// TwinCAT 3 PLC project PRG_Test_MachineControl
// ProgramVersion: 3.1.4024.0
// libraries:
//   B_Base, * (RafalOS)
//   B_IO, * (RafalOS)
//   B_MachineControl, * (RafalOS)
//   B_StatesAndModes, * (RafalOS)
//   Tc2_Standard, * (Beckhoff Automation GmbH)
//   Tc2_System, * (Beckhoff Automation GmbH)
//   Tc3_Module, * (Beckhoff Automation GmbH)
//   TcUnit, * (www.tcunit.org)
// project tree:
//   GVLs/ GVL_TopElement1.TcGVL (not stored), GVL_TopElement2.TcGVL (not stored), GVL_Variable.TcGVL
//   / PlcTask.TcTTO
//   POUs/ FB_MachineControlTest.TcPOU, FB_MyNewConfiguration.TcPOU
//   POUs/POUs TopElement1/ FB_ControlElement1.TcPOU, FB_ControlElement2.TcPOU, FB_TopElement1.TcPOU, ITF_ControlElement1.TcIO, ITF_ControlElement2.TcIO, ITF_TopElement1.TcIO
//   POUs/POUs TopElement2/ FB_ControlElement3.TcPOU, FB_ControlElement5.TcPOU (not stored), FB_ControlElement4.TcPOU, FB_ControlElement6.TcPOU (not stored), FB_GroupElement1.TcPOU (not stored), FB_TopElement2.TcPOU, ITF_ControlElement3.TcIO, ITF_ControlElement5.TcIO, ITF_ControlElement4.TcIO (not stored), ITF_ControlElement6.TcIO (not stored), ITF_GroupElement1.TcIO, ITF_TopElement2.TcIO
//   TESTs/ PRG_Test.TcPOU
// real-time tasks:
//   TASK PlcTask: cycle T#10ms, priority 20, ADS port 350

CONFIGURATION PRG_Test_MachineControl
    RESOURCE PLC ON TwinCAT3
        TASK PlcTask(INTERVAL := T#10ms, PRIORITY := 20);
        PROGRAM PRG_Test WITH PlcTask : PRG_Test;
    END_RESOURCE
END_CONFIGURATION

// ---- GVLs/GVL_Variable.TcGVL
{attribute 'qualified_only'}
VAR_GLOBAL
	fbMyNewConfiguration		: FB_MyNewConfiguration;
	
(* zmienne potrzebne do przetestowania samego SaMController	*)
	fbTime						: FB_BaseTime;
	fbLocation					: FB_BaseLocation;
	fbLogger					: FB_BaseLogger;
	stCommonData				: ST_BaseCommonData;
	flSS1						: FB_BaseFlag;
	flSTO						: FB_BaseFlag;
	fbMySaMController			: FB_SaMController;
END_VAR

// ---- POUs/POUs TopElement1/ITF_ControlElement1.TcIO
INTERFACE ITF_ControlElement1 EXTENDS ITF_BaseControlElement

END_INTERFACE

// ---- POUs/POUs TopElement1/ITF_ControlElement2.TcIO
INTERFACE ITF_ControlElement2 EXTENDS ITF_BaseControlElement

END_INTERFACE

// ---- POUs/POUs TopElement1/ITF_TopElement1.TcIO
INTERFACE ITF_TopElement1 EXTENDS ITF_BaseTopElement

END_INTERFACE

// ---- POUs/POUs TopElement2/ITF_ControlElement3.TcIO
INTERFACE ITF_ControlElement3 EXTENDS ITF_BaseControlElement

END_INTERFACE

// ---- POUs/POUs TopElement2/ITF_ControlElement5.TcIO
INTERFACE ITF_ControlElement5 EXTENDS ITF_BaseControlElement

END_INTERFACE

// ---- POUs/POUs TopElement2/ITF_GroupElement1.TcIO
INTERFACE ITF_GroupElement1 EXTENDS ITF_BaseGroupElement

END_INTERFACE

// ---- POUs/POUs TopElement2/ITF_TopElement2.TcIO
INTERFACE ITF_TopElement2 EXTENDS ITF_BaseTopElement

END_INTERFACE

// ---- TESTs/PRG_Test.TcPOU
PROGRAM PRG_Test
VAR
	fbSaMControllerTest				: FB_SaMControllerTest;
	fbMachineControlTest			: FB_MachineControl_NoneTE_Test;
	
END_VAR


	TcUnit.RUN_IN_SEQUENCE ();

END_PROGRAM

// ---- POUs/FB_MyNewConfiguration.TcPOU
FUNCTION_BLOCK FB_MyNewConfiguration EXTENDS FB_Base IMPLEMENTS ITF_Configuration
VAR

END_VAR

METHOD AddTopElementToLogger : BOOL
GVL_TopElement1.fbTopElement1.JoinTheLogger ();
GVL_TopElement2.fbTopElement2.JoinTheLogger ();
END_METHOD

(*			
	EVERDE sp. z o.o.
	Rafał Osajda		29.10.2025		TC 4024.66
	Dodawanie TopElementu do systemu
*)
METHOD AddTopElementToMachineControl : BOOL
VAR_INPUT
	itfMachineControl	: B_MachineControl.ITF_MachineControlConfigure;
END_VAR
THIS^.SetText (eLocation := E_BaseLocation.pl, wsDescription := "TopElement 1 pl");
THIS^.SetText (eLocation := E_BaseLocation.en, wsDescription := "TopElement 1 en");
THIS^.SetText (eLocation := E_BaseLocation.de, wsDescription := "TopElement 1 de");
GVL_TopElement1.fbTopElement1.SetName (stName := THIS^.GetTexts ());
itfMachineControl.AddTopElementFromConfiguration (fbTopElement	:= GVL_TopElement1.fbTopElement1);

THIS^.SetText (eLocation := E_BaseLocation.pl, wsDescription := "TopElement 2 pl");
THIS^.SetText (eLocation := E_BaseLocation.en, wsDescription := "TopElement 2 en");
THIS^.SetText (eLocation := E_BaseLocation.de, wsDescription := "TopElement 2 de");
GVL_TopElement1.fbTopElement1.SetName (stName := THIS^.GetTexts ());
itfMachineControl.AddTopElementFromConfiguration (fbTopElement	:= GVL_TopElement2.fbTopElement2);
END_METHOD

{warning 'add method implementation '}
METHOD SetStartMode : BOOL
VAR_INPUT
	itfMachineControl	: B_MachineControl.ITF_MachineControlConfigure;
END_VAR
END_METHOD

METHOD StateAndModes : BOOL
VAR_INPUT
	itfMachineControl	: B_MachineControl.ITF_MachineControlConfigure;
END_VAR
END_METHOD

END_FUNCTION_BLOCK

// ---- POUs/FB_MachineControlTest.TcPOU
FUNCTION_BLOCK FB_MachineControlTest EXTENDS TcUnit.FB_TestSuite
VAR

END_VAR


T01_TestPierwszegoPrzejscia ();
T02_TestInicjalizacjiSaM ();

METHOD PROTECTED T01_TestPierwszegoPrzejscia
VAR_INPUT
END_VAR
IF (TcUnit.TEST_ORDERED ('T01_TestPierwszegoPrzejscia')) THEN
	PRG_SystemControlMachineInit ();	//<- do prawdziwego programu
	AssertEquals_INT (Expected := 0, Actual := GVL_SystemVariable.fbMachineConfigure.iNubmerOfAddedConfigure, Message := 'T01_01 - blad ilosci konfiguracji');

	GVL_SystemVariable.fbMachineConfigure.AddConfiguration (fbConfigure := GVL_Variable.fbMyNewConfiguration); 		//<- do prawdziwego programu
	AssertEquals_INT (Expected := 1, Actual := GVL_SystemVariable.fbMachineConfigure.iNubmerOfAddedConfigure, Message := 'T01_02 - blad ilosci konfiguracji');

	PRG_SystemControlMachineWork ();		//<- do prawdziwego programu
	AssertTrue (Condition := GVL_SystemVariable.fbMachineControl.bInitializeCycle, Message := 'T02_01 - blad pierwszego przejscia');
	AssertTrue (Condition := GVL_SystemVariable.fbMachineControl.bInitDone, Message := 'T02_02 - blad inicjalizacji');
	AssertEquals_UINT (Expected := 20, Actual := GVL_SystemVariable.fbLogger.uiNumerOfReportsIntheSystem, Message := 'T02_03 - Bledna ilosc zgloszen');
	AssertEquals_UINT (Expected := 34, Actual := GVL_SystemVariable.fbMachineControl.uiNumberOfAllAddedElements, Message := 'T02_04 - bledna ilosc elementow');
	
	
	
	TcUnit.TEST_FINISHED ();
END_IF
END_METHOD

METHOD PROTECTED T02_TestInicjalizacjiSaM
VAR
	
END_VAR
IF (TcUnit.TEST_ORDERED ('T02_TestInicjalizacjiSaM')) THEN
	GVL_Variable.stCommonData.itfTime			:= GVL_Variable.fbTime;
	GVL_Variable.stCommonData.itfLocaciotn		:= GVL_Variable.fbLocation;
	GVL_Variable.stCommonData.itfLogger			:= GVL_Variable.fbLogger;
	GVL_Variable.fbMySaMController.LinkCommonData (stCommonData := GVL_Variable.stCommonData);
	GVL_Variable.fbMySaMController.LinkSS1 (fbSS1	:= GVL_Variable.flSS1);
	GVL_Variable.fbMySaMController.LinkSTO (fbSTO	:= GVL_Variable.flSTO);
	
	TcUnit.TEST_FINISHED ();
END_IF
END_METHOD

END_FUNCTION_BLOCK

// ---- POUs/POUs TopElement1/FB_ControlElement1.TcPOU
FUNCTION_BLOCK FB_ControlElement1 EXTENDS FB_BaseControlElement IMPLEMENTS ITF_ControlElement1
VAR
	
	itfsenStart			: ITF_IOSensor;
	itfsenEnd			: ITF_IOSensor;	
END_VAR

METHOD FB_init : BOOL
VAR_INPUT
	bInitRetains : BOOL; // if TRUE, the retain variables are initialized (warm start / cold start)
	bInCopyCode : BOOL;  // if TRUE, the instance afterwards gets moved into the copy code (online change)
	itfsenStart			: ITF_IOSensor;
	itfsenEnd			: ITF_IOSensor;	
	
END_VAR
THIS^.itfsenStart					:= itfsenStart;
THIS^.AddComponent (itfComponent	:= itfsenStart);
THIS^.SetText (eLocation 			:= E_BaseLocation.pl, wsDescription := "Nazwa komponentu 1 pl");
THIS^.SetText (eLocation 			:= E_BaseLocation.en, wsDescription := "Nazwa komponentu 1 en");
THIS^.SetText (eLocation 			:= E_BaseLocation.de, wsDescription := "Nazwa komponentu 1 de");
THIS^.itfsenStart.SetName (stName	:= THIS^.GetTexts ());

THIS^.itfsenEnd						:= itfsenEnd;
THIS^.AddComponent (itfComponent	:= itfsenEnd);
THIS^.SetText (eLocation 			:= E_BaseLocation.pl, wsDescription := "Nazwa komponentu 2 pl");
THIS^.SetText (eLocation 			:= E_BaseLocation.en, wsDescription := "Nazwa komponentu 2 en");
THIS^.SetText (eLocation 			:= E_BaseLocation.de, wsDescription := "Nazwa komponentu 2 de");
THIS^.itfsenEnd.SetName (stName	:= THIS^.GetTexts ());
END_METHOD

END_FUNCTION_BLOCK

// ---- POUs/POUs TopElement1/FB_ControlElement2.TcPOU
FUNCTION_BLOCK FB_ControlElement2 EXTENDS FB_BaseControlElement IMPLEMENTS ITF_ControlElement2
VAR
	
	itfsenStart			: ITF_IOSensor;
	itfsenEnd			: ITF_IOSensor;	
	itfsenPosition1		: ITF_IOSensor;	
	itfsenPosition2		: ITF_IOSensor;	
END_VAR

METHOD FB_init : BOOL
VAR_INPUT
	bInitRetains : BOOL; // if TRUE, the retain variables are initialized (warm start / cold start)
	bInCopyCode : BOOL;  // if TRUE, the instance afterwards gets moved into the copy code (online change)
	itfsenStart			: ITF_IOSensor;
	itfsenEnd			: ITF_IOSensor;	
	itfsenPosition1		: ITF_IOSensor;	
	itfsenPosition2		: ITF_IOSensor;	
END_VAR
THIS^.itfsenStart					:= itfsenStart;
THIS^.AddComponent (itfComponent	:= itfsenStart);
THIS^.SetText (eLocation 			:= E_BaseLocation.pl, wsDescription := "Nazwa komponentu 1 pl");
THIS^.SetText (eLocation 			:= E_BaseLocation.en, wsDescription := "Nazwa komponentu 1 en");
THIS^.SetText (eLocation 			:= E_BaseLocation.de, wsDescription := "Nazwa komponentu 1 de");
THIS^.itfsenStart.SetName (stName	:= THIS^.GetTexts ());

THIS^.itfsenEnd						:= itfsenEnd;
THIS^.AddComponent (itfComponent	:= itfsenEnd);
THIS^.SetText (eLocation 			:= E_BaseLocation.pl, wsDescription := "Nazwa komponentu 2 pl");
THIS^.SetText (eLocation 			:= E_BaseLocation.en, wsDescription := "Nazwa komponentu 2 en");
THIS^.SetText (eLocation 			:= E_BaseLocation.de, wsDescription := "Nazwa komponentu 2 de");
THIS^.itfsenEnd.SetName (stName	:= THIS^.GetTexts ());

THIS^.itfsenPosition1				:= itfsenPosition1;
THIS^.AddComponent (itfComponent	:= itfsenPosition1);
THIS^.SetText (eLocation 			:= E_BaseLocation.pl, wsDescription := "Nazwa komponentu 3 pl");
THIS^.SetText (eLocation 			:= E_BaseLocation.en, wsDescription := "Nazwa komponentu 3 en");
THIS^.SetText (eLocation 			:= E_BaseLocation.de, wsDescription := "Nazwa komponentu 3 de");
THIS^.itfsenPosition1.SetName (stName	:= THIS^.GetTexts ());

THIS^.itfsenPosition2				:= itfsenPosition2;
THIS^.AddComponent (itfComponent	:= itfsenPosition2);
THIS^.SetText (eLocation 			:= E_BaseLocation.pl, wsDescription := "Nazwa komponentu 4 pl");
THIS^.SetText (eLocation 			:= E_BaseLocation.en, wsDescription := "Nazwa komponentu 4 en");
THIS^.SetText (eLocation 			:= E_BaseLocation.de, wsDescription := "Nazwa komponentu 4 de");
THIS^.itfsenPosition2.SetName (stName	:= THIS^.GetTexts ());
END_METHOD

END_FUNCTION_BLOCK

// ---- POUs/POUs TopElement1/FB_TopElement1.TcPOU
FUNCTION_BLOCK FB_TopElement1 EXTENDS FB_BaseTopElement IMPLEMENTS ITF_TopElement1
VAR
	itfControlElement1		: ITF_ControlElement1;
	itfControlElement2		: ITF_ControlElement2;
	itfsenElementPosition1	: ITF_IOSensor;
	itfsenElementPosition2	: ITF_IOSensor;
END_VAR

METHOD FB_init : BOOL
VAR_INPUT
	bInitRetains : BOOL; // if TRUE, the retain variables are initialized (warm start / cold start)
	bInCopyCode : BOOL;  // if TRUE, the instance afterwards gets moved into the copy code (online change)
	itfControlElement1		: ITF_ControlElement1;
	itfControlElement2		: ITF_ControlElement2;
	itfsenElementPosition1	: ITF_IOSensor;
	itfsenElementPosition2	: ITF_IOSensor;
END_VAR
THIS^.itfControlElement1			:= itfControlElement1;
THIS^.AddComponent (itfComponent	:= itfControlElement1);
THIS^.SetText (eLocation 			:= E_BaseLocation.pl, wsDescription := "Nazwa controlelementu 1 pl");
THIS^.SetText (eLocation 			:= E_BaseLocation.en, wsDescription := "Nazwa controlelementu 1 en");
THIS^.SetText (eLocation 			:= E_BaseLocation.de, wsDescription := "Nazwa controlelementu 1 de");
THIS^.itfControlElement1.SetName (stName	:= THIS^.GetTexts ());

THIS^.itfControlElement2			:= itfControlElement2;
THIS^.AddComponent (itfComponent	:= itfControlElement2);
THIS^.SetText (eLocation 			:= E_BaseLocation.pl, wsDescription := "Nazwa controlelementu 2 pl");
THIS^.SetText (eLocation 			:= E_BaseLocation.en, wsDescription := "Nazwa controlelementu 2 en");
THIS^.SetText (eLocation 			:= E_BaseLocation.de, wsDescription := "Nazwa controlelementu 2 de");
THIS^.itfControlElement2.SetName (stName	:= THIS^.GetTexts ());

THIS^.itfsenElementPosition1		:= itfsenElementPosition1;
THIS^.AddComponent (itfComponent	:= itfsenElementPosition1);
THIS^.SetText (eLocation 			:= E_BaseLocation.pl, wsDescription := "Nazwa komponentu 1 pl");
THIS^.SetText (eLocation 			:= E_BaseLocation.en, wsDescription := "Nazwa komponentu 1 en");
THIS^.SetText (eLocation 			:= E_BaseLocation.de, wsDescription := "Nazwa komponentu 1 de");
THIS^.itfsenElementPosition1.SetName (stName	:= THIS^.GetTexts ());

THIS^.itfsenElementPosition2		:= itfsenElementPosition2;
THIS^.AddComponent (itfComponent	:= itfsenElementPosition2);
THIS^.SetText (eLocation 			:= E_BaseLocation.pl, wsDescription := "Nazwa komponentu 2 pl");
THIS^.SetText (eLocation 			:= E_BaseLocation.en, wsDescription := "Nazwa komponentu 2 en");
THIS^.SetText (eLocation 			:= E_BaseLocation.de, wsDescription := "Nazwa komponentu 2 de");
THIS^.itfsenElementPosition2.SetName (stName	:= THIS^.GetTexts ());
END_METHOD

END_FUNCTION_BLOCK

// ---- POUs/POUs TopElement2/FB_ControlElement3.TcPOU
FUNCTION_BLOCK FB_ControlElement3 EXTENDS FB_BaseControlElement IMPLEMENTS ITF_ControlElement3
VAR
	
	itfsenStart			: ITF_IOSensor;
	itfsenEnd			: ITF_IOSensor;	
END_VAR

METHOD FB_init : BOOL
VAR_INPUT
	bInitRetains : BOOL; // if TRUE, the retain variables are initialized (warm start / cold start)
	bInCopyCode : BOOL;  // if TRUE, the instance afterwards gets moved into the copy code (online change)
	itfsenStart			: ITF_IOSensor;
	itfsenEnd			: ITF_IOSensor;	
	
END_VAR
THIS^.itfsenStart					:= itfsenStart;
THIS^.AddComponent (itfComponent	:= itfsenStart);
THIS^.SetText (eLocation 			:= E_BaseLocation.pl, wsDescription := "Nazwa komponentu 1 pl");
THIS^.SetText (eLocation 			:= E_BaseLocation.en, wsDescription := "Nazwa komponentu 1 en");
THIS^.SetText (eLocation 			:= E_BaseLocation.de, wsDescription := "Nazwa komponentu 1 de");
THIS^.itfsenStart.SetName (stName	:= THIS^.GetTexts ());

THIS^.itfsenEnd						:= itfsenEnd;
THIS^.AddComponent (itfComponent	:= itfsenEnd);
THIS^.SetText (eLocation 			:= E_BaseLocation.pl, wsDescription := "Nazwa komponentu 2 pl");
THIS^.SetText (eLocation 			:= E_BaseLocation.en, wsDescription := "Nazwa komponentu 2 en");
THIS^.SetText (eLocation 			:= E_BaseLocation.de, wsDescription := "Nazwa komponentu 2 de");
THIS^.itfsenEnd.SetName (stName	:= THIS^.GetTexts ());
END_METHOD

END_FUNCTION_BLOCK

// ---- POUs/POUs TopElement2/FB_ControlElement4.TcPOU
FUNCTION_BLOCK FB_ControlElement4 EXTENDS FB_BaseControlElement IMPLEMENTS ITF_ControlElement4
VAR
	
	itfsenStart			: ITF_IOSensor;
	itfsenEnd			: ITF_IOSensor;	
	itfsenPosition1		: ITF_IOSensor;	
	itfsenPosition2		: ITF_IOSensor;	
END_VAR

METHOD FB_init : BOOL
VAR_INPUT
	bInitRetains : BOOL; // if TRUE, the retain variables are initialized (warm start / cold start)
	bInCopyCode : BOOL;  // if TRUE, the instance afterwards gets moved into the copy code (online change)
	itfsenStart			: ITF_IOSensor;
	itfsenEnd			: ITF_IOSensor;	
	itfsenPosition1		: ITF_IOSensor;	
	itfsenPosition2		: ITF_IOSensor;	
END_VAR
THIS^.itfsenStart					:= itfsenStart;
THIS^.AddComponent (itfComponent	:= itfsenStart);
THIS^.SetText (eLocation 			:= E_BaseLocation.pl, wsDescription := "Nazwa komponentu 1 pl");
THIS^.SetText (eLocation 			:= E_BaseLocation.en, wsDescription := "Nazwa komponentu 1 en");
THIS^.SetText (eLocation 			:= E_BaseLocation.de, wsDescription := "Nazwa komponentu 1 de");
THIS^.itfsenStart.SetName (stName	:= THIS^.GetTexts ());

THIS^.itfsenEnd						:= itfsenEnd;
THIS^.AddComponent (itfComponent	:= itfsenEnd);
THIS^.SetText (eLocation 			:= E_BaseLocation.pl, wsDescription := "Nazwa komponentu 2 pl");
THIS^.SetText (eLocation 			:= E_BaseLocation.en, wsDescription := "Nazwa komponentu 2 en");
THIS^.SetText (eLocation 			:= E_BaseLocation.de, wsDescription := "Nazwa komponentu 2 de");
THIS^.itfsenEnd.SetName (stName	:= THIS^.GetTexts ());

THIS^.itfsenPosition1				:= itfsenPosition1;
THIS^.AddComponent (itfComponent	:= itfsenPosition1);
THIS^.SetText (eLocation 			:= E_BaseLocation.pl, wsDescription := "Nazwa komponentu 3 pl");
THIS^.SetText (eLocation 			:= E_BaseLocation.en, wsDescription := "Nazwa komponentu 3 en");
THIS^.SetText (eLocation 			:= E_BaseLocation.de, wsDescription := "Nazwa komponentu 3 de");
THIS^.itfsenPosition1.SetName (stName	:= THIS^.GetTexts ());

THIS^.itfsenPosition2				:= itfsenPosition2;
THIS^.AddComponent (itfComponent	:= itfsenPosition2);
THIS^.SetText (eLocation 			:= E_BaseLocation.pl, wsDescription := "Nazwa komponentu 4 pl");
THIS^.SetText (eLocation 			:= E_BaseLocation.en, wsDescription := "Nazwa komponentu 4 en");
THIS^.SetText (eLocation 			:= E_BaseLocation.de, wsDescription := "Nazwa komponentu 4 de");
THIS^.itfsenPosition2.SetName (stName	:= THIS^.GetTexts ());
END_METHOD

END_FUNCTION_BLOCK

// ---- POUs/POUs TopElement2/FB_TopElement2.TcPOU
FUNCTION_BLOCK FB_TopElement2 EXTENDS FB_BaseTopElement IMPLEMENTS ITF_TopElement2
VAR
	itfGroupElement1		: ITF_GroupElement1;
	itfControlElement5		: ITF_ControlElement5;
	itfControlElement6		: ITF_ControlElement6;
	itfsenElementPosition1	: ITF_IOSensor;
	itfsenElementPosition2	: ITF_IOSensor;
END_VAR

METHOD FB_init : BOOL
VAR_INPUT
	bInitRetains : BOOL; // if TRUE, the retain variables are initialized (warm start / cold start)
	bInCopyCode : BOOL;  // if TRUE, the instance afterwards gets moved into the copy code (online change)
	itfGroupElement1		: ITF_GroupElement1;
	itfControlElement5		: ITF_ControlElement5;
	itfControlElement6		: ITF_ControlElement6;
	itfsenElementPosition1	: ITF_IOSensor;
	itfsenElementPosition2	: ITF_IOSensor;
END_VAR
THIS^.itfGroupElement1				:= itfGroupElement1;
THIS^.AddControlElement (itfControlElement	:= itfGroupElement1);
THIS^.SetText (eLocation 			:= E_BaseLocation.pl, wsDescription := "Nazwa group element 1 pl");
THIS^.SetText (eLocation 			:= E_BaseLocation.en, wsDescription := "Nazwa group element 1 en");
THIS^.SetText (eLocation 			:= E_BaseLocation.de, wsDescription := "Nazwa group element 1 de");
THIS^.itfGroupElement1.SetName (stName	:= THIS^.GetTexts ());

THIS^.itfControlElement5			:= itfControlElement5;
THIS^.AddControlElement (itfControlElement	:= itfControlElement5);
THIS^.SetText (eLocation 			:= E_BaseLocation.pl, wsDescription := "Nazwa controlelementu 1 pl");
THIS^.SetText (eLocation 			:= E_BaseLocation.en, wsDescription := "Nazwa controlelementu 1 en");
THIS^.SetText (eLocation 			:= E_BaseLocation.de, wsDescription := "Nazwa controlelementu 1 de");
THIS^.itfControlElement5.SetName (stName	:= THIS^.GetTexts ());

THIS^.itfControlElement6			:= itfControlElement6;
THIS^.AddControlElement (itfControlElement	:= itfControlElement6);
THIS^.SetText (eLocation 			:= E_BaseLocation.pl, wsDescription := "Nazwa controlelementu 2 pl");
THIS^.SetText (eLocation 			:= E_BaseLocation.en, wsDescription := "Nazwa controlelementu 2 en");
THIS^.SetText (eLocation 			:= E_BaseLocation.de, wsDescription := "Nazwa controlelementu 2 de");
THIS^.itfControlElement6.SetName (stName	:= THIS^.GetTexts ());

THIS^.itfsenElementPosition1		:= itfsenElementPosition1;
THIS^.AddComponent (itfComponent	:= itfsenElementPosition1);
THIS^.SetText (eLocation 			:= E_BaseLocation.pl, wsDescription := "Nazwa komponentu 1 pl");
THIS^.SetText (eLocation 			:= E_BaseLocation.en, wsDescription := "Nazwa komponentu 1 en");
THIS^.SetText (eLocation 			:= E_BaseLocation.de, wsDescription := "Nazwa komponentu 1 de");
THIS^.itfsenElementPosition1.SetName (stName	:= THIS^.GetTexts ());

THIS^.itfsenElementPosition2		:= itfsenElementPosition2;
THIS^.AddComponent (itfComponent	:= itfsenElementPosition2);
THIS^.SetText (eLocation 			:= E_BaseLocation.pl, wsDescription := "Nazwa komponentu 2 pl");
THIS^.SetText (eLocation 			:= E_BaseLocation.en, wsDescription := "Nazwa komponentu 2 en");
THIS^.SetText (eLocation 			:= E_BaseLocation.de, wsDescription := "Nazwa komponentu 2 de");
THIS^.itfsenElementPosition2.SetName (stName	:= THIS^.GetTexts ());
END_METHOD

END_FUNCTION_BLOCK
